// TIA Portal V20 export
DATA_BLOCK "Instance_FB_IO_Device_Functional_Test_Rework_DB"   // DB112
// stored: AutoNumber false, InstanceOfName FB_IO_Device_Functional_Test_Rework, InstanceOfType FB
"FB_IO_Device_Functional_Test_Rework"
   // VAR_INPUT
   //    Reset_PLC_Functional_Test_Rework : Bool;
   //    Status : Bool;
   //    Voltage_Read : UInt;
   //    Min_Electrical_Current : UInt;
   //    Max_Electrical_Current : UInt;
   //    Time_End_Electrical_Current_Test : Time;
   //    Time_Start_Visual_Test : Time;
   //    In_Functional_Test_Rework : "IO_Device_Functinal_Test_Rework";
   // END_VAR
   // VAR_OUTPUT
   //    Out_Test_Parameters_Rework : "IO_Device_Test_Parameters_Rework";
   //    Comunication_Error_Panel_Rework : Bool;
   // END_VAR
   // VAR
   //    Timer_Alarme_A_1 { S7_SetPoint := 'True'} : TON_TIME;
   //    Timer_Alarme_B_1 { S7_SetPoint := 'True'} : TON_TIME;
   // END_VAR
BEGIN
END_DATA_BLOCK
